// Mitsubishi GX Works2 project: 140630音声   PLC: FX1N/FX1NC

PROGRAM MAIN
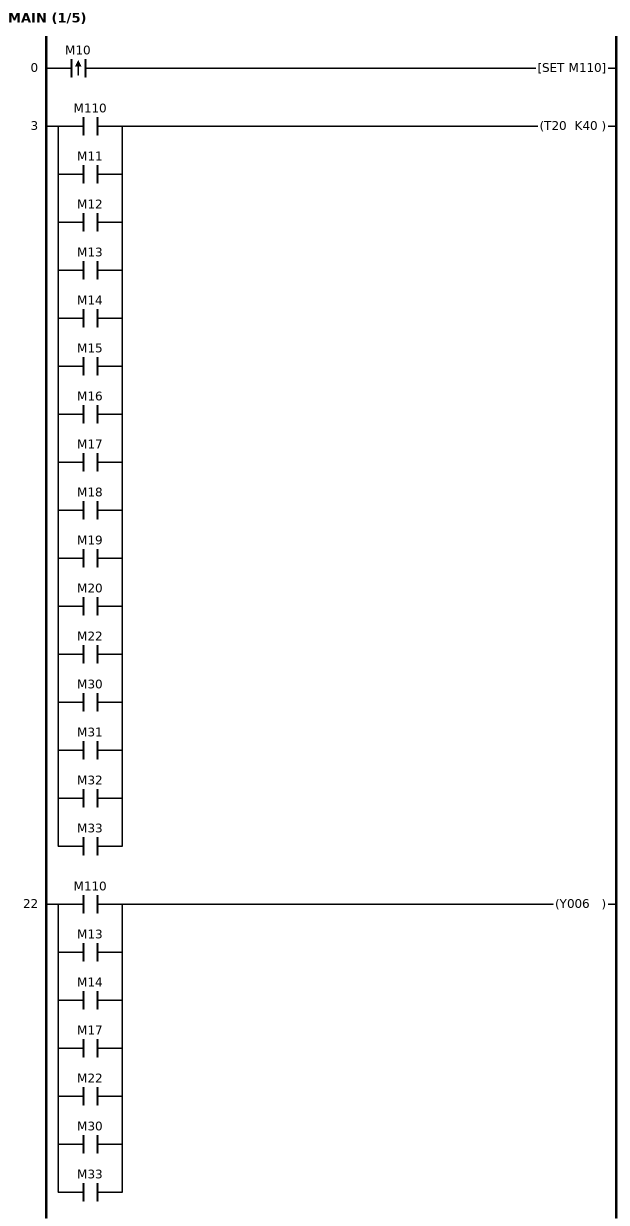
0     LDP     M10
      SET     M110
3     LD      M110
      OR      M11
      OR      M12
      OR      M13
      OR      M14
      OR      M15
      OR      M16
      OR      M17
      OR      M18
      OR      M19
      OR      M20
      OR      M22
      OR      M30
      OR      M31
      OR      M32
      OR      M33
      OUT     T20 K40
22    LD      M110
      OR      M13
      OR      M14
      OR      M17
      OR      M22
      OR      M30
      OR      M33
      OUT     Y006
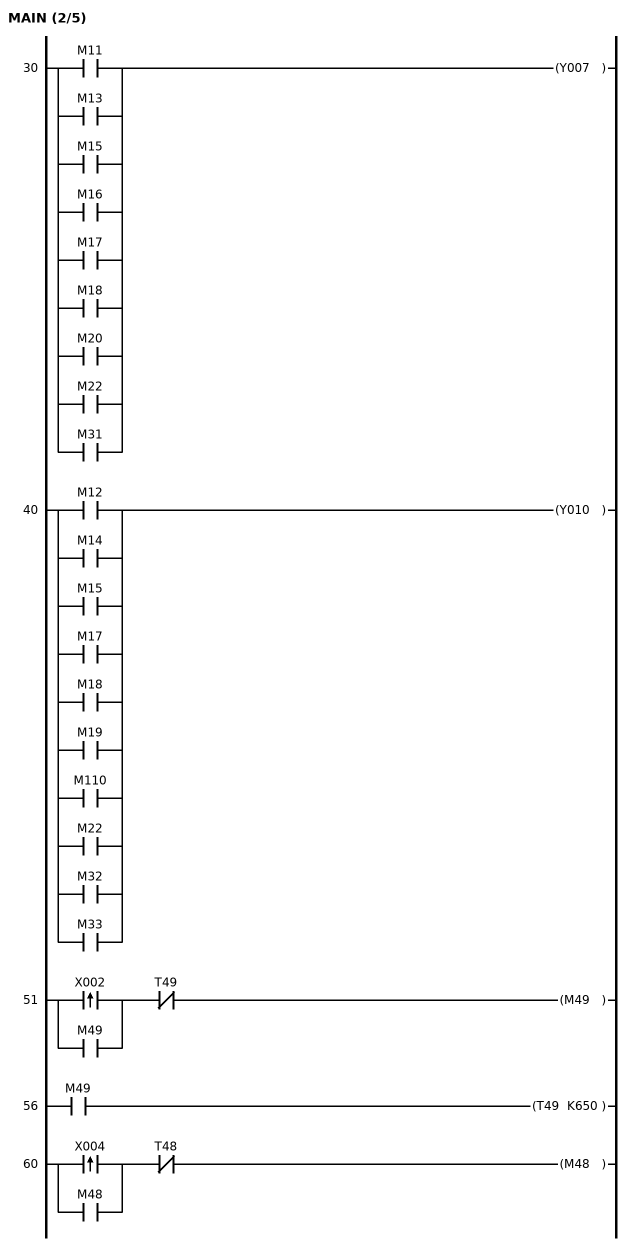
30    LD      M11
      OR      M13
      OR      M15
      OR      M16
      OR      M17
      OR      M18
      OR      M20
      OR      M22
      OR      M31
      OUT     Y007
40    LD      M12
      OR      M14
      OR      M15
      OR      M17
      OR      M18
      OR      M19
      OR      M110
      OR      M22
      OR      M32
      OR      M33
      OUT     Y010
51    LDP     X002
      OR      M49
      ANI     T49
      OUT     M49
56    LD      M49
      OUT     T49 K650
60    LDP     X004
      OR      M48
      ANI     T48
      OUT     M48
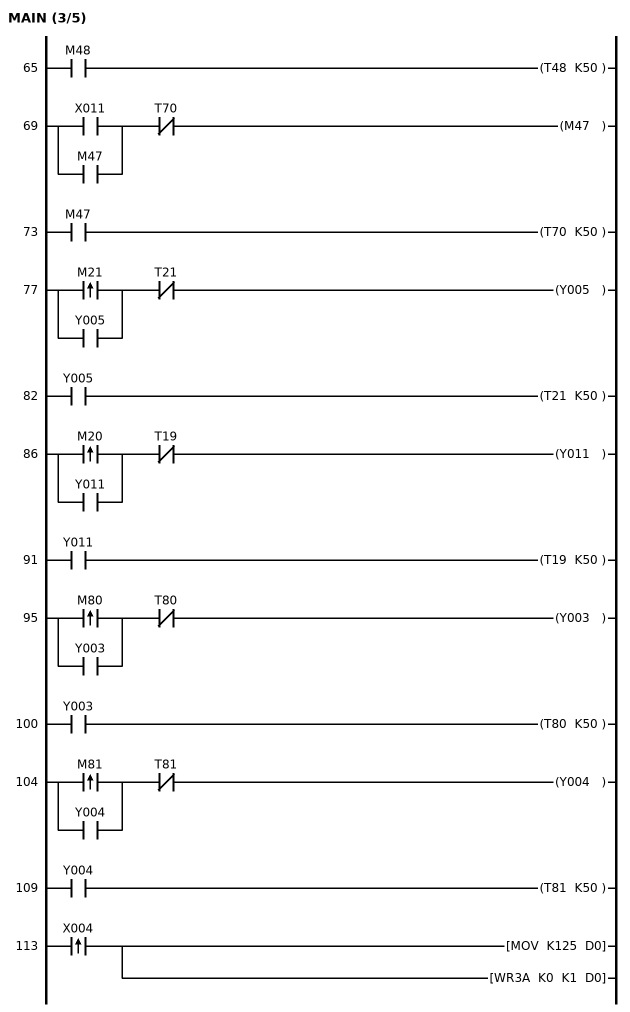
65    LD      M48
      OUT     T48 K50
69    LD      X011
      OR      M47
      ANI     T70
      OUT     M47
73    LD      M47
      OUT     T70 K50
77    LDP     M21
      OR      Y005
      ANI     T21
      OUT     Y005
82    LD      Y005
      OUT     T21 K50
86    LDP     M20
      OR      Y011
      ANI     T19
      OUT     Y011
91    LD      Y011
      OUT     T19 K50
95    LDP     M80
      OR      Y003
      ANI     T80
      OUT     Y003
100   LD      Y003
      OUT     T80 K50
104   LDP     M81
      OR      Y004
      ANI     T81
      OUT     Y004
109   LD      Y004
      OUT     T81 K50
113   LDP     X004
      MOV     K125 D0
      WR3A    K0 K1 D0
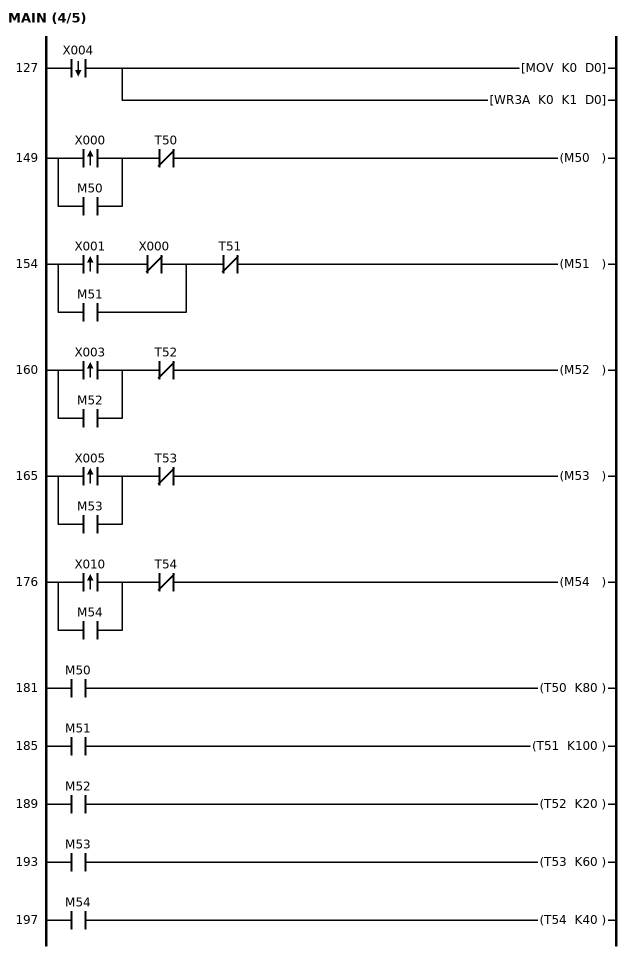
127   LDF     X004
      MOV     K0 D0
      WR3A    K0 K1 D0
149   LDP     X000
      OR      M50
      ANI     T50
      OUT     M50
154   LDP     X001
      ANI     X000
      OR      M51
      ANI     T51
      OUT     M51
160   LDP     X003
      OR      M52
      ANI     T52
      OUT     M52
165   LDP     X005
      OR      M53
      ANI     T53
      OUT     M53
176   LDP     X010
      OR      M54
      ANI     T54
      OUT     M54
181   LD      M50
      OUT     T50 K80
185   LD      M51
      OUT     T51 K100
189   LD      M52
      OUT     T52 K20
193   LD      M53
      OUT     T53 K60
197   LD      M54
      OUT     T54 K40
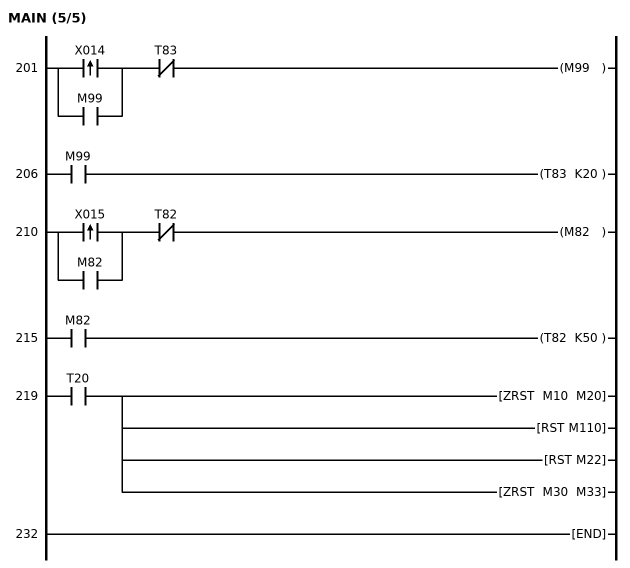
201   LDP     X014
      OR      M99
      ANI     T83
      OUT     M99
206   LD      M99
      OUT     T83 K20
210   LDP     X015
      OR      M82
      ANI     T82
      OUT     M82
215   LD      M82
      OUT     T82 K50
219   LD      T20
      ZRST    M10 M20
      RST     M110
      RST     M22
      ZRST    M30 M33
232   END
END_PROGRAM
